// Mitsubishi GX Works2 project: PLC RS485   PLC: FX3U/FX3UC

PROGRAM MAIN
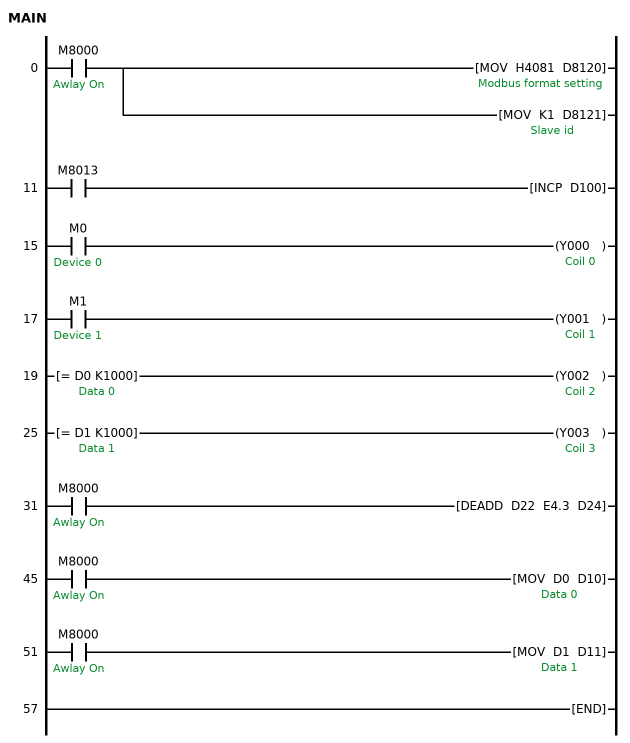
0     LD      M8000  ; Awlay On
      MOV     H4081 D8120  ; Modbus format setting
      MOV     K1 D8121  ; Slave id
11    LD      M8013
      INCP    D100
15    LD      M0  ; Device 0
      OUT     Y000  ; Coil 0
17    LD      M1  ; Device 1
      OUT     Y001  ; Coil 1
19    LD=     D0 K1000  ; Data 0
      OUT     Y002  ; Coil 2
25    LD=     D1 K1000  ; Data 1
      OUT     Y003  ; Coil 3
31    LD      M8000  ; Awlay On
      DEADD   D22 E4.3 D24
45    LD      M8000  ; Awlay On
      MOV     D0 D10
51    LD      M8000  ; Awlay On
      MOV     D1 D11
57    END
END_PROGRAM
